// TIA Portal V18 export
DATA_BLOCK "SS1_770A1_16DO_DO_Vars"   // DB11072
{ S7_Optimized_Access := 'FALSE' }
VERSION : 0.1
// stored: AutoNumber false, DBAccessibleFromOPCUA true, IsOnlyStoredInLoadMemory false, IsWriteProtectedInAS false
   VAR
      DO1 { S7_SetPoint := 'True'} : "UDT_DOadv";   // Резерв
      DO2 { S7_SetPoint := 'True'} : "UDT_DOadv";   // Резерв
      DO3 { S7_SetPoint := 'True'} : "UDT_DOadv";   // Вкл. тепл. вент (8.x)
      DO4 { S7_SetPoint := 'True'} : "UDT_DOadv";   // HS Вкл. насос (10.203)
      DO5 { S7_SetPoint := 'True'} : "UDT_DOadv";   // HS Вкл. насос (10.202)
      DO6 { S7_SetPoint := 'True'} : "UDT_DOadv";   // HS Дозвіл на роботу пальник 1- ст. К1
      DO7 { S7_SetPoint := 'True'} : "UDT_DOadv";   // HS Дозвіл на роботу пальник 2- ст. К1
      DO8 { S7_SetPoint := 'True'} : "UDT_DOadv";   // AHU NF Вкл. цирк. насос (2.202)
      DO9 { S7_SetPoint := 'True'} : "UDT_DOadv";   // AHU NF Дозвіл на роботу 1- ст. ККБ
      DO10 { S7_SetPoint := 'True'} : "UDT_DOadv";   // AHU NF Дозвіл на роботу 2- ст. ККБ
      DO11 { S7_SetPoint := 'True'} : "UDT_DOadv";   // AHU NF Дозвіл на роботу 3- ст. ККБ
      DO12 { S7_SetPoint := 'True'} : "UDT_DOadv";   // AHU NF Дозвіл на роботу 4- ст. ККБ
      DO13 { S7_SetPoint := 'True'} : "UDT_DOadv";   // AHU NF Вкл. 1- шв. пр. вент. (2.200)
      DO14 { S7_SetPoint := 'True'} : "UDT_DOadv";   // AHU NF Вкл. 2- шв. пр. вент. (2.200)
      DO15 { S7_SetPoint := 'True'} : "UDT_DOadv";   // HS Дозвіл на роботу пальник 1- ст. К2
      DO16 { S7_SetPoint := 'True'} : "UDT_DOadv";   // HS Дозвіл на роботу пальник 2- ст. К2
   END_VAR
BEGIN
   DO1.iFuncSystemID := 10;
   DO1.iFuncVar := 10;
   DO2.iFuncSystemID := 10;
   DO2.iFuncVar := 11;
   DO3.iFuncSystemID := 10;
   DO3.iFuncVar := 12;
   DO4.iFuncSystemID := 100;
   DO4.iFuncVar := 1;
   DO5.iFuncSystemID := 100;
   DO5.iFuncVar := 5;
   DO6.iFuncSystemID := 100;
   DO6.iFuncVar := 3;
   DO7.iFuncSystemID := 10;
   DO7.iFuncVar := 5;
   DO8.iFuncSystemID := 10;
   DO8.iFuncVar := 6;
   DO9.iFuncSystemID := 10;
   DO9.iFuncVar := 13;
   DO14.iFuncSystemID := 1;
   DO14.iFuncVar := 1;
   DO14.cMOA := 1;
   DO15.iFuncSystemID := 1;
   DO16.iFuncSystemID := 1;
   DO16.iFuncVar := 3;
END_DATA_BLOCK
